{attribute 'qualified_only'}
VAR_GLOBAL
	DateTime: DATE_AND_TIME;
END_VAR

(* stored: Version 1.1.0.1, ProductVersion 3.1.4024.0
   GVL Gen: Id {4a5c7f26-a090-4482-a00e-1e80d8c2ab58} *)
